// TIA Portal V20 export
TYPE "typeSequenceControlNodeJobInterface_jrOutPnPLeft"
// stored: Namespace Unit1.Em2
   STRUCT
      stack1PICKJob2 : "LER_typeJobInterface";
      stack2PICKJob3 : "LER_typeJobInterface";
      PLACEJob4 : "LER_typeJobInterface";
   END_STRUCT;
END_TYPE
